// Retrieves the number of PLC tasks available in the system.
FUNCTION F_GetNumberOfPlcTasks : T_Size // The number of PLC tasks.

F_GetNumberOfPlcTasks := SIZEOF(TwinCAT_SystemInfoVarList._TaskInfo) / SIZEOF(PlcTaskSystemInfo);

END_FUNCTION

(* stored: Version 1.1.0.1
   POU F_GetNumberOfPlcTasks: Id {8dac3619-28ef-094c-37c8-ea1d77a553b6}, SpecialFunc None *)
